{attribute 'linkalways'} 
{attribute 'no_explicit_call' := 'This FB is a CLASS and must be accessed using methods or properties'}
{attribute 'enable_dynamic_creation'}
{attribute 'hide_all_locals'}
FUNCTION_BLOCK ABSTRACT Node EXTENDS Disposable IMPLEMENTS I_Node
VAR
	_id : T_MAXSTRING;
	_order : DINT;
	_mode : DINT;
	eventEmitter : EventEmitter;
	inputPortHost : InputPortHost(THIS^, eventEmitter);
	outputPortHost : OutputPortHost(THIS^, eventEmitter);
	parameterHost : ParameterHost(THIS^, eventEmitter);
	contentHost : ContentHost(THIS^, eventEmitter);
	alarmHost : AlarmHost(THIS^, eventEmitter);
	metadataHost : MetadataHost(THIS^, eventEmitter);
	extensionHost : ExtensionHost(THIS^,eventEmitter);
	deserializationFailedAlarm : DeserializationFailedAlarm(THIS^);
END_VAR

METHOD PUBLIC Accept
VAR_INPUT
	Visitor : I_NodeVisitor;
END_VAR
Visitor.VisitNode(THIS^);
END_METHOD

METHOD PROTECTED AddContent : I_Content
VAR_INPUT
	Name : T_MAXSTRING;
	Data : I_Datatype;
END_VAR
AddContent := Contents.AddDataAsContent(Name, Data);
END_METHOD

METHOD PROTECTED AddInput : I_InputPort
VAR_INPUT
	Name : T_MAXSTRING;
	Data : I_Datatype;
END_VAR
AddInput := InputPorts.AddDataAsInputPort(Name, Data);
END_METHOD

METHOD PUBLIC AddMetadata : I_HostMetadata
VAR_INPUT
	Name : T_MAXSTRING;
	Data : I_Datatype;
END_VAR
Metadatum.AddDataAsMetadata(Name, Data);
AddMetadata := THIS^;
END_METHOD

METHOD PROTECTED AddOutput : I_OutputPort
VAR_INPUT
	Name : T_MAXSTRING;
	Data : I_Datatype;
END_VAR
AddOutput := OutputPorts.AddDataAsOutputPort(Name, Data);
END_METHOD

METHOD PROTECTED AddParameter : I_Parameter
VAR_INPUT
	Name : T_MAXSTRING;
	Data : I_Datatype;
END_VAR
AddParameter := Parameters.AddDataAsParameter(Name, Data);
END_METHOD

PROPERTY PUBLIC Alarms : I_Alarms
GET
Alarms := alarmHost;
END_GET
END_PROPERTY

METHOD PRIVATE CheckIfNodeExecutionIsBlocked : BOOL;
VAR
	nodePreExecuteEvent : NodePreExecuteEvent(THIS^);
END_VAR
eventEmitter.Emit('OnNodePreExecute',nodePreExecuteEvent);
CheckIfNodeExecutionIsBlocked := nodePreExecuteEvent.ExecuteCancelled;
END_METHOD

METHOD PUBLIC ABSTRACT Clone : I_Node
VAR_INPUT
END_VAR
END_METHOD

PROPERTY PUBLIC Contents : I_Contents
GET
Contents := contentHost;
END_GET
END_PROPERTY

METHOD PRIVATE EmitNodeExecuteBeginEvent : BOOL;
VAR
	nodeExecuteBeginEvent : NodeExecuteBeginEvent(THIS^);
END_VAR
eventEmitter.Emit('OnNodeExecuteBegin',nodeExecuteBeginEvent);
END_METHOD

METHOD PRIVATE EmitNodeExecuteEndEvent : BOOL;
VAR
	nodeExecuteEndEvent : NodeExecuteEndEvent(THIS^);
END_VAR
eventEmitter.Emit('OnNodeExecuteEnd',nodeExecuteEndEvent);
END_METHOD

METHOD PUBLIC Execute
IF CheckIfNodeExecutionIsBlocked() THEN
	RETURN;
END_IF

EmitNodeExecuteBeginEvent();
OnExecute();
EmitNodeExecuteEndEvent();
END_METHOD

PROPERTY PUBLIC Extensions : I_Extensions
GET
Extensions := extensionHost;
END_GET
END_PROPERTY

PROPERTY PUBLIC HasRaisedAlarm : BOOL
GET
HasRaisedAlarm := alarmHost.HasRaisedAlarm;
END_GET
END_PROPERTY

PROPERTY PUBLIC Id : T_MAXSTRING
GET
Id := _id;
END_GET
END_PROPERTY

PROPERTY PUBLIC InputPorts : I_InputPorts
GET
InputPorts := inputPortHost;
END_GET
END_PROPERTY

PROPERTY PUBLIC Metadatum : I_Metadatum
GET
Metadatum := metadataHost;
END_GET
END_PROPERTY

PROPERTY PUBLIC Mode : DINT
GET
Mode := _mode;
END_GET
END_PROPERTY

METHOD PUBLIC OffEvent
VAR_INPUT
	EventName : T_MaxString;
	EventHandler : I_EventHandler;
END_VAR
eventEmitter.OffEvent(EventName, EventHandler);
END_METHOD

METHOD PUBLIC OnceEvent
VAR_INPUT
	EventName : T_MaxString;
	EventHandler : I_EventHandler;
END_VAR
eventEmitter.OnceEvent(EventName, EventHandler);
END_METHOD

METHOD PUBLIC OnEvent
VAR_INPUT
	EventName : T_MaxString;
	EventHandler : I_EventHandler;
END_VAR
eventEmitter.OnEvent(EventName, EventHandler);
END_METHOD

METHOD PROTECTED ABSTRACT OnExecute : HRESULT
END_METHOD

PROPERTY PUBLIC Order : DINT
GET
Order := _order;
END_GET
END_PROPERTY

PROPERTY PUBLIC OutputPorts : I_OutputPorts
GET
OutputPorts := outputPortHost;
END_GET
END_PROPERTY

PROPERTY PUBLIC Parameters : I_Parameters
GET
Parameters := parameterHost;
END_GET
END_PROPERTY

PROPERTY PUBLIC Self : I_Node
GET
Self := This^;
END_GET
END_PROPERTY

METHOD PUBLIC SerializeWith
VAR_INPUT
	Serializer : I_Serializer;
END_VAR
Serializer.StartObject();
Serializer.AddKeyString('id',_id);
Serializer.AddKeyDint('order',_order);
Serializer.AddKeyDint('mode',_mode);
inputPortHost.SerializeWith(Serializer);
outputPortHost.SerializeWith(Serializer);
parameterHost.SerializeWith(Serializer);
contentHost.SerializeWith(Serializer);
alarmHost.SerializeWith(Serializer);
extensionHost.SerializeWith(Serializer);
metadataHost.SerializeWith(Serializer);
Serializer.EndObject();
END_METHOD

METHOD PUBLIC TryDeserializeFrom : BOOL
VAR_INPUT
	Deserializer : I_Deserializer;
	Feedback : I_DeserializerFeedback;
END_VAR
DeserializationFailedAlarm.Clear();

IF NOT Deserializer.TryGetKeyString('id', _id, Feedback) THEN
	DeserializationFailedAlarm.Raise('Missing node id');	
	RETURN;
END_IF

IF NOT Deserializer.TryGetKeyDint('order', _order, Feedback) THEN
	DeserializationFailedAlarm.Raise('Missing node order');	
	RETURN;
END_IF

IF NOT Deserializer.TryGetKeyDint('mode', _mode, Feedback) THEN
	DeserializationFailedAlarm.Raise('Missing node mode');	
	RETURN;
END_IF

IF NOT parameterHost.TryDeserializeFrom(Deserializer, Feedback) THEN
	DeserializationFailedAlarm.Raise('Failed to deserialize parameters');	
	RETURN;
END_IF

IF NOT extensionHost.TryDeserializeFrom(Deserializer, Feedback) THEN
	DeserializationFailedAlarm.Raise('Failed to deserialize extensions');	
	RETURN;
END_IF

TryDeserializeFrom := TRUE;
END_METHOD

END_FUNCTION_BLOCK

(* stored: Version 1.1.0.1, ProductVersion 3.1.4024.13
   POU Node: Id {dea4a6e6-88e8-4a03-84ea-b39393a5373f}, SpecialFunc None
   Folder Abstract: Id {8193ee30-b78d-4ea0-bfbe-c2a5814340d9}
   Folder Private: Id {b58aec16-127f-40f3-807e-1336c1cce4cc}
   Folder Protected: Id {b89c0aab-4104-081c-26ed-eda79ec1f8c0}
   Method Accept: Id {dd7a8e72-4444-4df2-b876-dec7f4fae19f}
   Method AddContent: Id {f94bf07c-731b-0ce4-1bdc-49a7103a3255}
   Method AddInput: Id {0475b747-7d7c-0bc9-13ae-202f2a6a0841}
   Method AddMetadata: Id {7537f1c9-8f79-00b5-1961-3ebfa452305f}
   Method AddOutput: Id {d2ca7345-1329-099c-256e-314ef745dda3}
   Method AddParameter: Id {f55d9acc-06d9-0fdf-37f0-cff1f3e0aecb}
   Property Alarms: Id {f0a6c976-17db-4461-8af3-623f6953058b}
   Get Get: Id {011e7dea-c711-4aab-8fe6-920c2a083dc5}
   Method CheckIfNodeExecutionIsBlocked: Id {e6c90d14-caf8-469c-8e84-a87816f43889}
   Method Clone: Id {864cba3a-3ba1-492d-b1fd-367b7ddeeac3}
   Property Contents: Id {043f0496-9047-4c55-a014-a217d44038a6}
   Get Get: Id {82d4143b-5313-4d9b-a102-f6756ed3e4aa}
   Method EmitNodeExecuteBeginEvent: Id {77ca6a46-059c-4018-b367-fa23a314306c}
   Method EmitNodeExecuteEndEvent: Id {a42b5b3b-ff9d-471e-a9b1-7e26b88f78ad}
   Method Execute: Id {53111ca4-ff22-4d20-85e1-3d604fc86fe1}
   Property Extensions: Id {d2cfced0-e0d5-465c-bcc4-ce23e7f52568}
   Get Get: Id {2659ad4f-3e76-4c6d-8fd3-7d40632c166f}
   Property HasRaisedAlarm: Id {4249ccf7-b508-431a-9ef2-e1a366472d7e}
   Get Get: Id {488e699a-a946-49fc-97e6-db19d62c0c4c}
   Property Id: Id {63f297b4-8bc6-432b-9391-959282b386ac}
   Get Get: Id {c7cddb10-45f3-4cb1-94e1-6c7bf991fee1}
   Property InputPorts: Id {667e2ef4-8314-4f08-b4e3-05a0e645d26e}
   Get Get: Id {600fe8c7-2deb-41f2-a84d-75775139cb4d}
   Property Metadatum: Id {dc1c33ab-3c00-4382-a179-94135e27aa02}
   Get Get: Id {c5fb408d-4da2-4d29-9876-e015636ab2f5}
   Property Mode: Id {f3a4ecf5-6aa2-4420-a695-7b91c1e23089}
   Get Get: Id {ca53613b-1735-4175-9d85-7543ddd08da7}
   Method OffEvent: Id {be27ce50-cd40-41ee-ba8b-d8a27b92e94e}
   Method OnceEvent: Id {44098522-81d9-4a99-b4fa-7682f4e2c6aa}
   Method OnEvent: Id {9f6ebfb1-fc41-4f9a-a9e6-3469f96c80ea}
   Method OnExecute: Id {f0f0499a-5f72-4d57-9065-48b06559724d}
   Property Order: Id {0ad930d6-e597-400e-905a-66b1d732b9fb}
   Get Get: Id {688751d6-d2ec-49a7-a744-ad796dd65c51}
   Property OutputPorts: Id {0fbd802c-e4d8-449d-9fbb-541b4b378024}
   Get Get: Id {4fc89f54-cd65-48c8-a4b8-5d34cce1154c}
   Property Parameters: Id {0b68b859-b935-4386-9545-23a9d1985319}
   Get Get: Id {d9e95db6-d150-4bed-aaa7-83500b4095f9}
   Property Self: Id {d0638425-cacb-415b-9410-d46817128d19}
   Get Get: Id {6f132944-1e78-41dc-953b-8c04f1cf77ef}
   Method SerializeWith: Id {0900fa8f-2c1c-4681-b602-0d226a708c72}
   Method TryDeserializeFrom: Id {feda9c40-f82c-4c3a-b07d-cecee9133921} *)
